Yaskawa INFORM job: R1_W45-48(90,0)KM-OK.JBI

/JOB
//NAME R1_W45-48(90,0)KM-OK
///FOLDERNAME KRIS-SCIANA
//POS
///NPOS 87,87,0,6,0,0
///TOOL 0
///POSTYPE PULSE
///PULSE
C00000=-614,-36100,-109393,1002,105622,-76266
C00001=-614,-36100,-109393,1002,105622,-76266
C00002=30112,-127063,-118472,-9266,74977,-65479
C00003=146783,-41222,-44528,-14508,92298,-23932
C00004=177758,-18432,-24897,-15900,96897,-12902
C00005=166847,35431,29185,-16026,89350,-15768
C00006=166321,37118,32341,-15327,88247,-16677
C00007=166321,37589,33997,-15328,87496,-16584
C00008=166321,37118,32341,-15327,88247,-16677
C00009=171699,4841,-760,-15279,92918,-15369
C00010=170835,-35200,-22324,-18799,58263,-10772
C00011=166066,-33100,-15421,-17623,54185,-12058
C00012=165910,-32536,-14743,-17588,54031,-12098
C00013=165593,-31712,-14199,-17442,54048,-12239
C00014=167025,-37605,-22579,-17571,56389,-12034
C00015=161139,-1958,-5557,-939,83085,-16350
C00016=160390,25614,20531,-865,81188,-16590
C00017=160390,25904,21696,-866,80621,-16587
C00018=160640,27890,23636,-893,80451,-16499
C00019=160390,25457,19886,-865,81505,-16593
C00020=160390,25655,20697,-865,81108,-16591
C00021=160390,25965,21925,-866,80512,-16587
C00022=160390,25906,21695,-866,80622,-16587
C00023=160724,27768,23517,-901,80463,-16471
C00024=160390,25446,19834,-865,81532,-16594
C00025=165643,13675,12551,-10985,79337,-20135
C00026=167674,10013,12505,-14753,77464,-21361
C00027=167674,10387,13747,-14782,76911,-21293
C00028=167674,10317,13522,-14776,77011,-21304
C00029=167700,12673,15637,-14783,76929,-21284
C00030=167674,9804,11798,-14735,77782,-21397
C00031=161667,10120,9793,-4034,79193,-25528
C00032=160919,6459,2756,-3926,81599,-25861
C00033=171280,-20527,-2481,-28534,71438,2255
C00034=169873,-15007,4957,-28696,69425,2217
C00035=167060,-14489,6711,-28588,67760,1526
C00036=167060,-13749,8427,-28718,67162,1682
C00037=167060,-14037,7762,-28667,67393,1622
C00038=166465,-12361,9034,-28595,67262,1417
C00039=167060,-14860,5838,-28526,68066,1445
C00040=165078,-24102,-3856,-28103,68483,543
C00041=174496,-24787,-5330,-32767,69285,4466
C00042=172819,-19212,1769,-32913,67371,4356
C00043=172173,-16914,4714,-32988,66590,4329
C00044=171876,-16211,5234,-32949,66511,4228
C00045=171876,-15504,6876,-33099,65965,4402
C00046=171876,-15676,6480,-33063,66097,4360
C00047=171337,-14366,7462,-32993,65949,4178
C00048=171876,-15676,6480,-33063,66097,4360
C00049=161265,-34405,-11426,-23449,56557,-2204
C00050=165693,-30942,-7306,-24884,57138,-447
C00051=166684,-37324,-14511,-24847,58482,-354
C00052=186406,-34667,3928,-73065,39460,-38715
C00053=184274,-31936,5659,-72637,38187,-39290
C00054=183554,-30919,6459,-72582,37731,-39429
C00055=184413,-32109,5553,-72669,38270,-39251
C00056=183286,-31712,4384,-71496,37848,-40087
C00057=183702,-30600,6752,-72608,37823,-39394
C00058=184249,-31903,5681,-72632,38172,-39297
C00059=186379,-34635,3948,-73060,39445,-38722
C00060=167722,9367,7612,-23360,62585,-34243
C00061=167801,13027,10888,-23414,62483,-34188
C00062=167142,16072,13321,-23174,62357,-34430
C00063=167756,12648,9658,-23288,62989,-34316
C00064=167388,13497,12126,-23376,61886,-34228
C00065=173332,10285,11302,-25598,62601,-31933
C00066=172874,7418,5891,-25066,64150,-32484
C00067=172893,3803,2763,-25059,64217,-32492
C00068=164197,30117,28508,-7284,75788,-59159
C00069=159404,38154,42543,-9157,72246,-60449
C00070=167377,18214,26493,-16202,68026,18911
C00071=167619,17632,26517,-16279,67773,19037
C00072=156382,28059,35230,8276,60397,-62214
C00073=156516,28450,35749,8244,60265,-62173
C00074=158228,21529,30144,8085,56459,-62151
C00075=169524,15489,24358,3475,55983,-57295
C00076=169990,15192,24251,3294,55877,-57113
C00077=171015,11241,21938,1424,52896,-56666
C00078=171426,9412,20997,657,51671,-56465
C00079=171094,8446,20464,813,51503,-56607
C00080=171378,-10003,-1750,645,55690,-56461
C00081=177862,-30287,-28528,4670,80588,-54952
C00082=118728,-111618,-84953,4597,80939,-55645
C00083=93138,-143334,-112968,-11263,80414,-55836
C00084=69157,-157081,-130798,3838,14431,-65536
C00085=4993,-152746,-129686,-4359,15988,-61765
C00086=4993,-152746,-129686,-14331,-5080,-57274
BC00000=263312,1241177,821509
BC00001=263312,1190158,821509
BC00002=346073,1190032,739965
BC00003=373252,1189540,420639
BC00004=380468,1189409,335861
BC00005=380509,1189408,335374
BC00006=380509,1189408,335374
BC00007=380509,1189408,335374
BC00008=380509,1189408,335374
BC00009=380509,1189408,335374
BC00010=380509,1189408,335374
BC00011=380509,1189408,335374
BC00012=380509,1189408,335374
BC00013=380509,1189408,335374
BC00014=380509,1189408,335374
BC00015=380509,1189408,335374
BC00016=380509,1189408,335374
BC00017=380509,1189408,335374
BC00018=380509,1189408,335374
BC00019=380509,1189408,335374
BC00020=380509,1189408,335374
BC00021=380509,1189408,335374
BC00022=380509,1189408,335374
BC00023=380509,1189408,335374
BC00024=380509,1189408,335374
BC00025=360576,1190661,359570
BC00026=352914,1191142,368871
BC00027=352914,1191142,368871
BC00028=352914,1191142,368871
BC00029=352914,1191142,368871
BC00030=352914,1191142,368871
BC00031=352914,1191142,368871
BC00032=352914,1191142,368871
BC00033=314729,1191142,414305
BC00034=314729,1191142,414305
BC00035=314729,1191142,414305
BC00036=314729,1191142,414305
BC00037=314729,1191142,414305
BC00038=314729,1191142,414305
BC00039=314729,1191142,414305
BC00040=314729,1191142,414305
BC00041=342456,1191142,396778
BC00042=342456,1191142,396778
BC00043=342456,1191142,396778
BC00044=342456,1191142,396778
BC00045=342456,1191142,396778
BC00046=342456,1191142,396778
BC00047=342456,1191142,396778
BC00048=342456,1191142,396778
BC00049=342456,1191142,396778
BC00050=342456,1191142,396778
BC00051=342456,1191142,396778
BC00052=380947,1191142,366768
BC00053=380218,1191142,346373
BC00054=379927,1191142,338215
BC00055=379927,1191142,338215
BC00056=379927,1191142,338215
BC00057=347389,1191142,339098
BC00058=347681,1191142,347256
BC00059=348410,1191142,367652
BC00060=395053,1191142,340155
BC00061=395053,1191142,316827
BC00062=395053,1191142,307496
BC00063=395053,1191142,307496
BC00064=395053,1191142,307496
BC00065=395053,1191142,307496
BC00066=395053,1191142,300232
BC00067=395053,1191142,323560
BC00068=393354,1191142,386943
BC00069=393354,1191142,386943
BC00070=373050,1191142,387415
BC00071=373050,1191142,387415
BC00072=393354,1191142,386943
BC00073=393354,1191142,386943
BC00074=393354,1191142,386943
BC00075=393354,1191142,386943
BC00076=393354,1191142,386943
BC00077=393354,1191142,386943
BC00078=393354,1191142,386943
BC00079=393354,1191142,386943
BC00080=393354,1191142,386943
BC00081=393355,1191142,386938
BC00082=393355,1191142,386938
BC00083=393355,1191142,1007665
BC00084=338999,1191026,1023031
BC00085=1321,1191026,1023031
BC00086=1321,699716,1054830
///POSTYPE BASE
///RECTAN
///RCONF 0,0,0,0,0,0,0,0,0,0,0,0,0,0,0,0,0,0,0,0,0,0,0,0
P00006=0.222,-3.123,-1.508,0.0000,0.0000,0.0000
P00023=0.143,-0.036,0.682,0.0000,0.0000,0.0000
P00024=0.145,-0.552,1.326,0.0000,0.0000,0.0000
P00026=0.562,-0.002,-0.337,0.0000,0.0000,0.0000
P00027=-0.746,0.015,-9.096,0.0000,0.0000,0.0000
P00030=5.926,-4.294,-1.390,0.0000,0.0000,0.0000
//INST
///DATE 2024/07/30 08:31
///ATTR SC,RW
///GROUP1 RB1,BS1
NOP
'r1_W45-48(90,0)
'Path S904
SFTOF
MOVJ C00000 BC00000 VJ=100.00
MOVJ C00001 BC00001 VJ=100.00
MOVJ C00002 BC00002 VJ=100.00
MOVJ C00003 BC00003 VJ=100.00
MOVJ C00004 BC00004 VJ=100.00
MOVL C00005 BC00005 V=166.7
MOVL C00006 BC00006 V=60.0
REFP 3 C00007 BC00007
CALL JOB:SEARCH-R1
SET P026 P006
SFTON P026
MOVL C00008 BC00008 V=60.0
MOVL C00009 BC00009 V=133.3
MOVL C00010 BC00010 V=133.3
MOVL C00011 BC00011 V=133.3
MOVL C00012 BC00012 V=60.0
REFP 3 C00013 BC00013
CALL JOB:SEARCH-R1
SET P026 P006
SFTON P026
MOVL C00014 BC00014 V=100.0
MOVL C00015 BC00015 V=133.3
MOVL C00016 BC00016 V=100.0
MOVL C00017 BC00017 V=60.0
REFP 3 C00018 BC00018
CALL JOB:SEARCH-R1
SET P026 P006
SFTON P026
MOVL C00019 BC00019 V=60.0
'Path S902
SFTOF
MOVL C00020 BC00020 V=60.0
REFP 3 C00021 BC00021
CALL JOB:SEARCH-R1
SET P030 P006
SFTON P030
MOVL C00022 BC00022 V=60.0
REFP 3 C00023 BC00023
CALL JOB:SEARCH-R1
SET P030 P006
SFTON P030
MOVL C00024 BC00024 V=60.0
MOVL C00025 BC00025 V=166.7
MOVL C00026 BC00026 V=60.0
REFP 3 C00027 BC00027
CALL JOB:SEARCH-R1
SET P024 P006
SFTON P024
MOVL C00028 BC00028 V=60.0
REFP 3 C00029 BC00029
CALL JOB:SEARCH-R1
SET P024 P006
SFTON P024
MOVL C00030 BC00030 V=60.0
MOVL C00031 BC00031 V=166.7
MOVL C00032 BC00032 V=166.7
'Path S901
SFTOF
MOVJ C00033 BC00033 VJ=100.00
MOVJ C00034 BC00034 VJ=100.00
MOVL C00035 BC00035 V=60.0
REFP 3 C00036 BC00036
CALL JOB:SEARCH-R1
SET P023 P006
SFTON P023
MOVL C00037 BC00037 V=60.0
REFP 3 C00038 BC00038
CALL JOB:SEARCH-R1
SET P023 P006
SFTON P023
MOVL C00039 BC00039 V=60.0
MOVL C00040 BC00040 V=166.7
'Path S1151
SFTOF
MOVJ C00041 BC00041 VJ=100.00
MOVJ C00042 BC00042 VJ=100.00
MOVL C00043 BC00043 V=100.0
MOVL C00044 BC00044 V=60.0
REFP 3 C00045 BC00045
CALL JOB:SEARCH-R1
SET P027 P006
SFTON P027
MOVL C00046 BC00046 V=60.0
REFP 3 C00047 BC00047
CALL JOB:SEARCH-R1
SET P027 P006
SFTON P027
MOVL C00048 BC00048 V=60.0
MOVL C00049 BC00049 V=100.0
MOVL C00050 BC00050 V=166.7
MOVL C00051 BC00051 V=166.7
'Path W467
SFTOF
SFTON P027
MOVJ C00052 BC00052 VJ=100.00
MOVJ C00053 BC00053 VJ=100.00
MOVL C00054 BC00054 V=100.0 PL=0
REFP 1 C00055 BC00055
REFP 2 C00056 BC00056
MACRO1 MJ#(0) ARGF9
ARCON
SFTON P023
MOVL C00057 BC00057 V=10.0
ARCOF
MOVL C00058 BC00058 V=166.7
MOVL C00059 BC00059 V=166.7
SFTOF
SFTON P026
MOVJ C00060 BC00060 VJ=100.00
MOVJ C00061 BC00061 VJ=100.00
MOVL C00062 BC00062 V=100.0 PL=0
REFP 1 C00063 BC00063
REFP 2 C00064 BC00064
MACRO1 MJ#(0) ARGF6
ARCON
WVON WEV#(40)
MOVL C00065 BC00065 V=7.5
ARCOF
WVOF
MOVL C00066 BC00066 V=166.7
MACRO1 MJ#(0) ARGF9
MOVL C00067 BC00067 V=166.7
SFTOF
'Path W474
SFTON P026
MOVJ C00068 BC00068 VJ=100.00
MOVL C00069 BC00069 V=100.0 PL=0
REFP 1 C00070 BC00070
REFP 2 C00071 BC00071
MACRO1 MJ#(0) ARGF6
ARCON
WVON WEV#(40)
MOVL C00072 BC00072 V=7.5
MOVL C00073 BC00073 V=7.5
WVOF
MACRO1 MJ#(0) ARGF9
SFTON P030
MOVL C00074 BC00074 V=10.0
SFTON P024
MOVL C00075 BC00075 V=10.0
MOVL C00076 BC00076 V=10.0
MOVL C00077 BC00077 V=10.0
MOVL C00078 BC00078 V=10.0
MOVL C00079 BC00079 V=10.0
ARCOF
SFTOF
MOVL C00080 BC00080 V=100.0
MOVL C00081 BC00081 V=166.7
MOVJ C00082 BC00082 VJ=100.00
MOVJ C00083 BC00083 VJ=100.00
MOVJ C00084 BC00084 VJ=100.00
MOVJ C00085 BC00085 VJ=100.00
MOVJ C00086 BC00086 VJ=100.00
SFTOF
END
